FUNCTION_BLOCK FB_Latch
VAR_INPUT
	setState		:BOOL;
	resetState		:BOOL;
END_VAR
VAR_OUTPUT
	output			:BOOL;
	invertOutput	:Bool;
END_VAR
VAR
END_VAR

output := NOT(resetState OR invertOutput);

invertOutput := NOT (setState OR output);

END_FUNCTION_BLOCK

(* stored: Version 1.1.0.1, ProductVersion 3.1.4024.12
   POU FB_Latch: Id {87088223-f9b4-435b-94c2-28d259e49779}, SpecialFunc None *)
